TYPE ST_G120_Control :
STRUCT
	bSafetyOk			: BOOL;
	bRun				: BOOL;
	bClearFault			: BOOL;
	nSpeedHz 			: UINT;
	bInvertDirection		: BOOL;
END_STRUCT
END_TYPE

(* stored: Version 1.1.0.1, ProductVersion 3.1.4024.15
   DUT ST_G120_Control: Id {86a9cc3c-2485-4ab8-a74f-be737fde4c57} *)
